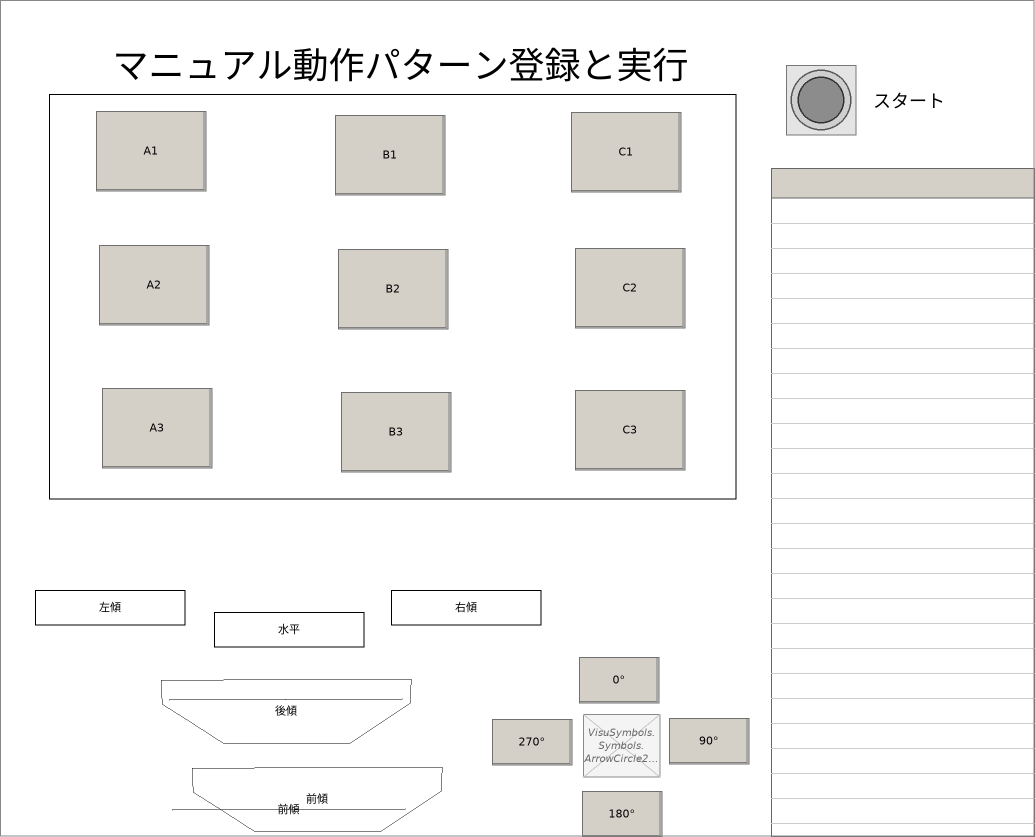
VISUALIZATION Visualization_recipe  // 1035x837
    RoundedRectangle (49,94 687x405)
    Button (575,390 110x80), "C3"
        tap MAIN.manupilator_buttons[8]
    Button (575,248 110x80), "C2"
        tap MAIN.manupilator_buttons[7]
    Button (571,112 110x80), "C1"
        tap MAIN.manupilator_buttons[6]
    Button (335,115 110x80), "B1"
        tap MAIN.manupilator_buttons[5]
    Button (338,249 110x80), "B2"
        tap MAIN.manupilator_buttons[4] p3779583253=TRUE
    Button (341,392 110x80), "B3"
        tap MAIN.manupilator_buttons[3]
    Button (96,111 110x80), "A1"
        tap MAIN.manupilator_buttons[2]
    Button (99,245 110x80), "A2"
        tap MAIN.manupilator_buttons[1]
    Button (102,388 110x80), "A3"
        tap MAIN.manupilator_buttons[0]
    Polyline (44,593) (45,594)
    RoundedRectangle (35,590 150x35), angle 330, "左傾"
        tap MAIN.manupilator_buttons[14] p3779583253=TRUE
    RoundedRectangle (391,590 150x35), angle 30, "右傾"
        tap MAIN.manupilator_buttons[13]
    Polygon (161,680) (411,679) (410,703) (350,743) (223,743) (189,721) (162,704), "後傾"
        tap MAIN.manupilator_buttons[12]
    Polyline (402,699) (169,700)
    Polygon (192,768) (442,767) (441,791) (381,831) (254,831) (220,809) (193,792), "前傾"
        tap MAIN.manupilator_buttons[11] p3779583253=TRUE
    Polyline (405,809) (172,810), "前傾"
    Table (771,168 264x669), data array: MAIN.Recipe_Display
        p3854506369: MAIN.Recipe_Display[INDEX]
        p2232123230: 登録処理内容
        p1128707560: bajp_jobmgmt.ParamFuturesLib.MAX_TASK_NUM
    Label (94,42 613x47), "マニュアル動作パターン登録と実行"
    PushSwitch (786,65 70x70), variable: MAIN.manual_start, behaviour: TAP, style: Switch-PushSwitch-Gray
    Label (868,78 82x47), "スタート"
    RoundedRectangle (214,612 150x35), "水平"
        tap MAIN.manupilator_buttons[15]
    Image (583,714 77x63), image: VisuSymbols.Symbols.ArrowCircle2LeftRightLeft
    Button (492,719 80x46), "270°"
        tap MAIN.manupilator_buttons[16]
    Button (579,657 80x46), "0°"
        tap MAIN.manupilator_buttons[17]
    Button (669,718 80x46), "90°"
        tap MAIN.manupilator_buttons[18]
    Button (582,791 80x46), "180°"
        tap MAIN.manupilator_buttons[19]
END_VISUALIZATION

(* stored: Version 1.1.0.1, ProductVersion 3.1.4024.12
   Visu Visualization_recipe: Id {df7e6850-0022-4037-9766-3e9fa19b1acf} *)
